FUNCTION_BLOCK CHECKPOINT_DISCOVERY_CAT (* Composite Function Block Type *)
  (* Standard: 61499-2 *)
  (* Version 0.0, 1/24/2023, Dmitrii, Flexbridge AB, template *)
  PACKAGE UAO.Hackathon;
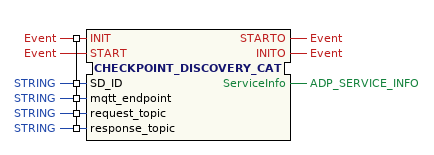
  EVENT_INPUT
    INIT WITH SD_ID, mqtt_endpoint, request_topic, response_topic;
    START;
  END_EVENT
  EVENT_OUTPUT
    STARTO;
    INITO;
  END_EVENT
  VAR_INPUT
    SD_ID : STRING;
    mqtt_endpoint : STRING;
    request_topic : STRING;
    response_topic : STRING;
  END_VAR
  PLUGS
    ServiceInfo : ADP_SERVICE_INFO;
  END_PLUGS
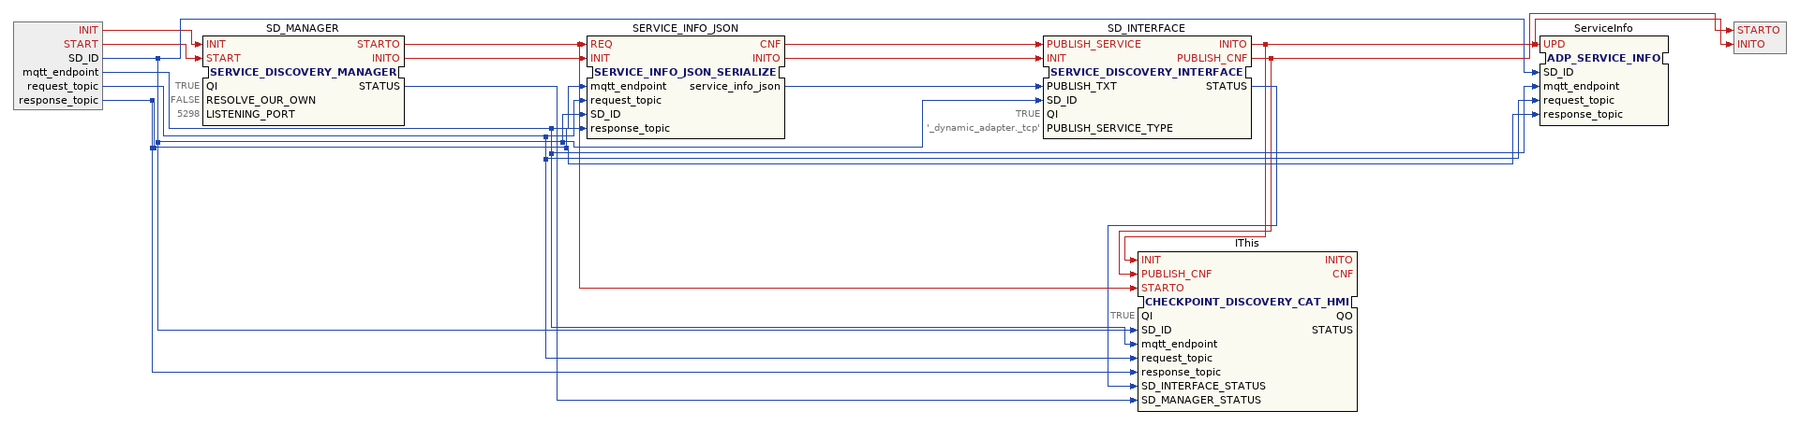
  FBS
    SD_INTERFACE : SERVICE_DISCOVERY_INTERFACE(QI := TRUE, PUBLISH_SERVICE_TYPE := '_dynamic_adapter._tcp');
    SD_MANAGER : SERVICE_DISCOVERY_MANAGER(QI := TRUE, RESOLVE_OUR_OWN := FALSE, LISTENING_PORT := 5298);
    SERVICE_INFO_JSON : SERVICE_INFO_JSON_SERIALIZE;
    IThis : CHECKPOINT_DISCOVERY_CAT_HMI(QI := TRUE);
  END_FBS
  EVENT_CONNECTIONS
    INIT TO SD_MANAGER.INIT;
    SD_INTERFACE.INITO TO INITO;
    SD_MANAGER.STARTO TO SERVICE_INFO_JSON.REQ;
    SERVICE_INFO_JSON.CNF TO SD_INTERFACE.PUBLISH_SERVICE;
    SD_MANAGER.INITO TO SERVICE_INFO_JSON.INIT;
    SERVICE_INFO_JSON.INITO TO SD_INTERFACE.INIT;
    START TO SD_MANAGER.START;
    SD_INTERFACE.INITO TO ServiceInfo.UPD;
    SD_INTERFACE.PUBLISH_CNF TO STARTO;
    SD_INTERFACE.INITO TO IThis.INIT;
    SD_INTERFACE.PUBLISH_CNF TO IThis.PUBLISH_CNF;
    SD_MANAGER.STARTO TO IThis.STARTO;
  END_CONNECTIONS
  DATA_CONNECTIONS
    mqtt_endpoint TO SERVICE_INFO_JSON.mqtt_endpoint;
    request_topic TO SERVICE_INFO_JSON.request_topic;
    SERVICE_INFO_JSON.service_info_json TO SD_INTERFACE.PUBLISH_TXT;
    SD_ID TO SERVICE_INFO_JSON.SD_ID;
    SD_ID TO ServiceInfo.SD_ID;
    SD_ID TO SD_INTERFACE.SD_ID;
    mqtt_endpoint TO ServiceInfo.mqtt_endpoint;
    request_topic TO ServiceInfo.request_topic;
    response_topic TO SERVICE_INFO_JSON.response_topic;
    response_topic TO ServiceInfo.response_topic;
    SD_ID TO IThis.SD_ID;
    mqtt_endpoint TO IThis.mqtt_endpoint;
    request_topic TO IThis.request_topic;
    response_topic TO IThis.response_topic;
    SD_INTERFACE.STATUS TO IThis.SD_INTERFACE_STATUS;
    SD_MANAGER.STATUS TO IThis.SD_MANAGER_STATUS;
  END_CONNECTIONS
END_FUNCTION_BLOCK
